{region '#Template'}
	{attribute 'Version' := '1.0.0.0'}
	{attribute 'Tags' := '"LCID": "1031", "Text": "H, Heating circuit, HtgCir, Setpoint"'}
	{attribute 'Tags' := '"LCID": "1033", "Text": "H, Heating circuit, HtgCir, Setpoint"'}
	{attribute 'Description' := '"LCID": "1031", "Text": "Sollwert Heizkreis"'}
	{attribute 'Description' := '"LCID": "1033", "Text": "Setpoint heating circuit"'}
{endregion}
FUNCTION_BLOCK FB_BA_H_HtgCir_Sp EXTENDS FB_BA_View
VAR_INPUT
	eOpMod					: E_BA_EnergyLvl;
	fSpFrstProtec			: REAL;
	fTWthDamp				: REAL;
END_VAR
VAR_OUTPUT
	fSpFlWT							: REAL;
END_VAR
VAR_INPUT CONSTANT
	NgtOffs					: FB_BA_AV_Op;	
	SpFlWT					: FB_BA_AV_Op;		
	HtgCrv					: FB_BA_Scale_04; 
END_VAR
VAR
	PrioSwi					: FB_BA_MMUX_R04;
END_VAR

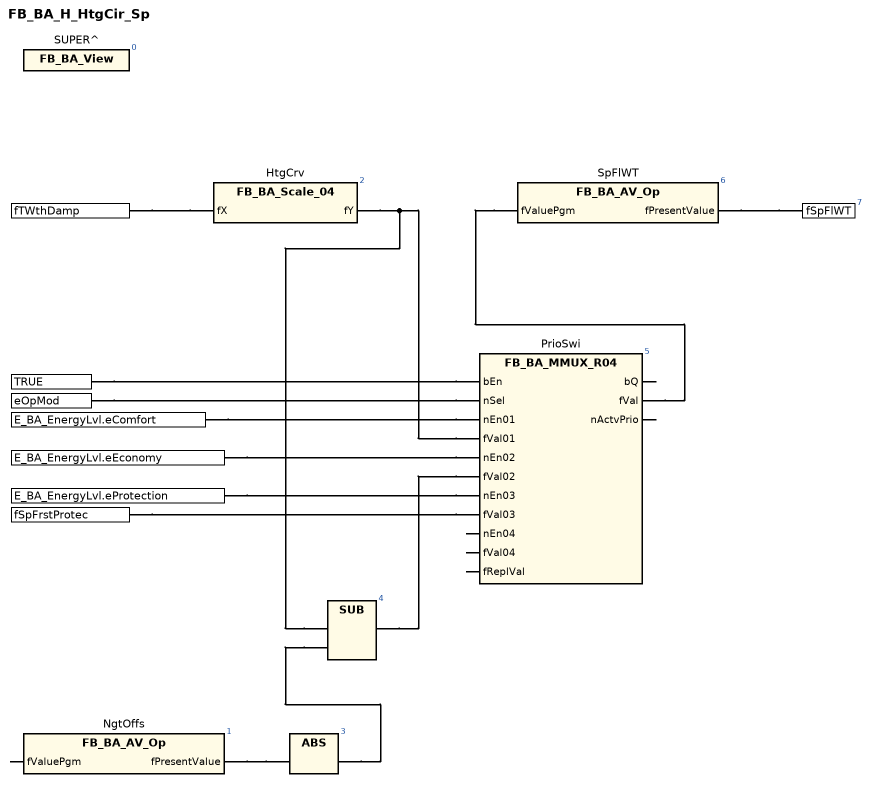
// note: 1 stored wires end on pins the file does not list and are not shown
SUPER^(); // FB_BA_View
NgtOffs(); // FB_BA_AV_Op
HtgCrv(fX := fTWthDamp); // FB_BA_Scale_04
PrioSwi(
    bEn := TRUE,
    nSel := eOpMod,
    nEn01 := E_BA_EnergyLvl.eComfort,
    fVal01 := HtgCrv.fY,
    nEn02 := E_BA_EnergyLvl.eEconomy,
    fVal02 := HtgCrv.fY - ABS(NgtOffs.fPresentValue),
    nEn03 := E_BA_EnergyLvl.eProtection,
    fVal03 := fSpFrstProtec); // FB_BA_MMUX_R04
SpFlWT(fValuePgm := PrioSwi.fVal); // FB_BA_AV_Op
fSpFlWT := SpFlWT.fPresentValue;

METHOD FB_init : BOOL
VAR_INPUT
	bInitRetains : BOOL; // if TRUE, the retain variables are initialized (warm start / cold start)
	bInCopyCode : BOOL;  // if TRUE, the instance afterwards gets moved into the copy code (online change)
END_VAR
NgtOffs.iParent				:= THIS^;
NgtOffs.iLabel				:= LblCmpHeating.H_HtgCir_Sp_NgtOffs;		 
NgtOffs.sObjectName			:= '{Idx=01}';
NgtOffs.eUnit				:= E_BA_Unit.eTemperature_DegreesCelsius;  
NgtOffs.fValueRm			:= 8.0;
NgtOffs.fCOVIncrement	:= BA2_Param.fDefCOVIncrement;							

SpFlWT.iParent				:= THIS^;
SpFlWT.iLabel				:= LblCmpHeating.H_HtgCir_Sp_SpFlWT;		 
SpFlWT.sObjectName			:= '{Idx=01}';
SpFlWT.eUnit				:= E_BA_Unit.eTemperature_DegreesCelsius;  
SpFlWT.fCOVIncrement		:= BA2_Param.fDefCOVIncrement;							

HtgCrv.iParent				:= THIS^;										
HtgCrv.iLabel				:= LblCmpHeating.H_HtgCir_Sp_HtgCrv;
HtgCrv.sObjectName			:= '{Idx=01}';										 
HtgCrv.eDPADMode			:= E_BA_DPADMode.eIncludeDescription; 
HtgCrv.X1.fValueRm			:= 15.0;
HtgCrv.X2.fValueRm			:= 0.0;
HtgCrv.X3.fValueRm			:= -10.0;
HtgCrv.X4.fValueRm			:= -20.0;
HtgCrv.Y1.fValueRm			:= 25.0;
HtgCrv.Y2.fValueRm			:= 40.0;
HtgCrv.Y3.fValueRm			:= 55.0;
HtgCrv.Y4.fValueRm			:= 65.0;
HtgCrv.YMin.fValueRm		:= 5.0;
HtgCrv.YMax.fValueRm		:= 80.0;
END_METHOD

END_FUNCTION_BLOCK

(* stored: Version 1.1.0.1, ProductVersion 3.1.4024.9
   POU FB_BA_H_HtgCir_Sp: Id {4674a590-cd7b-4f08-a48e-d8ce41368e14}, SpecialFunc None
   Method FB_init: Id {428a2269-79ea-4887-bd6e-ee7d5ba83bfd} *)
